# EPICS autosave request: iocBoot/iocTomoScan_2ID_STEP/auto_settings.req
file "tomoScan_settings.req", P=$(P), R=$(R)
file "tomoScan_step_settings.req", P=$(P), R=$(R)
file "tomoScan_2ID_settings.req", P=$(P), R=$(R)
